(* CODESYS project Cartesin.export

Project tree, tasks and I/O mapping:
  program Cartesin [ST]
*)

// Cartesin
PROGRAM Cartesin
VAR
	Enable : BOOL;
	StartMov : BOOL;
	safe_pos :  ARRAY [1..6] OF REAL := [0.0, 0.0, 0.0, 0.0, -90.0, 0.0];
	FirstReachPos :  ARRAY [1..6] OF REAL := [0.4, 0.1, 0.606, 180, 180.000, -0.0];
	SecondReachPos :  ARRAY [1..6] OF REAL := [0.4, -0.1, 0.606, 180, 180.000, -0.0];
	FirstPerPos :  ARRAY [1..6] OF REAL := [0.4, 0.1, 0.636, 180, 180.000, -0.0];
	SecondPerPos :  ARRAY [1..6] OF REAL := [0.4, -0.1, 0.636, 180, 180.000, -0.0];
	
	CurrentPos : REAL;
	Vel : REAL := 0.5;
	Acc : REAL := 1.5;
	Jerk : REAL := 4.5;
	safepoint_overfeed : INT := 5; 
	GrRelCorner :REAL := 0.5;
	MovGroup : INT := 0;
	
	MovErr : BOOL;
	
	PowBlk : AuxAxis_PowerOn;
	PowDone, PowErr : BOOL;
	
	MovState : INT;
	InitialMov : ArcaLibrary.MCAT_MoveDirect;;
	Movs : ARRAY [0..6] OF ArcaLibrary.MC_MoveLinearAbsolute;
	StopMov : ArcaLibrary.MC_GroupStop;
	dis_trig : r_trig;
	stopEnb: BOOL;
	
	// six axis IO, Button function management
	DIp : Digital_Input;
	DOp : Digital_Output;
	enb_Timer : ton;
	enb_Delay_Time : TIME := T#1S;
	
END_VAR

// IO management
Dip(enable := TRUE);
DOP(enable := TRUE);

IF dip.DI_01 THEN	// enb button manage
	enb_Timer(in:= TRUE, pt := enb_Delay_Time); // if button has been push more then 2s
	IF enb_timer.Q AND NOT enable THEN	// enable robot
		enb_Timer(in:= FALSE);
		enable := TRUE;
	ELSIF enb_timer.Q AND enable THEN	// disable robot
		enb_Timer(in:= FALSE);
		enable := FALSE;
	END_IF
ELSE
	enb_Timer(in:= FALSE);
END_IF

IF dip.DI_02 THEN // if start button has been pressed then start mov robot
	startMov := TRUE;
END_IF

IF NOT dip.DI_03 THEN // if stop button has been pressed then stop move robot
	startMov := FALSE;
END_IF

DOp(DO_07 := PowDone);	// if robot enabled then light on

PowBlk(Enable := enable, done => PowDone);

dis_trig(clk := NOT startMov);
IF dis_trig.Q THEN
	stopEnb := TRUE;
END_IF
StopMov(AxesGroup := MovGroup, execute := stopEnb AND NOT stopmov.Done, Deceleration := vel*100, jerk := vel*1000, BufferMode := mcAborting);
IF stopmov.Done OR NOT enable THEN
	stopEnb := FALSE;	
END_IF

IF MovState > 20 AND NOT startMov THEN
	MovState := 20;
END_IF

CASE MovState OF
	0:
		IF PowDone THEN
			MovState := 10;
		END_IF
	10:
		IF startMov THEN
			MovState := 20;
		END_IF
	20:
		InitialMov(axesgroup := MovGroup, execute := FALSE);
		Movs[0](axesgroup := MovGroup, Execute := FALSE);
		Movs[1](axesgroup := MovGroup, Execute := FALSE);
		Movs[2](axesgroup := MovGroup, Execute := FALSE);
		Movs[3](axesgroup := MovGroup, Execute := FALSE);
		Movs[4](axesgroup := MovGroup, Execute := FALSE);
		Movs[5](axesgroup := MovGroup, Execute := FALSE);
		IF startMov THEN
			MovState := 30;
		ELSE
			MovState := 0;
		END_IF
	30:
		InitialMov(axesgroup := MovGroup, execute := TRUE, position := ADR(safe_pos), coordsystem := mcacs
			, BufferMode:=mcAborting, TransitionMode:= tmNone, TransitionParameter:= ADR(GrRelCorner) 
			, OverFeedPerc:= safepoint_overfeed);
		IF initialmov.Done THEN
			MovState := 40;
		END_IF
	40:
		IF Movs[4].Done THEN
			Movs[5](axesgroup := MovGroup, Execute := TRUE, Position := ADR(SecondPerPos)
				, Velocity := vel, Acceleration := acc, Deceleration := Acc, jerk := jerk
				, coordsystem := mcMcs, BufferMode := mcBlendingNext
				, TransitionMode := TMcornerdistance, TransitionParameter:=ADR(GrRelCorner)
				, Error => MovErr);
		END_IF
		Movs[0](axesgroup := MovGroup, Execute := TRUE, Position := ADR(FirstPerPos)
			, Velocity := vel, Acceleration := acc, Deceleration := Acc, jerk := jerk
			, coordsystem := mcMcs, BufferMode := mcBlendingNext
			, TransitionMode := TMcornerdistance, TransitionParameter:=ADR(GrRelCorner)
			, Error => MovErr);
		Movs[1](axesgroup := MovGroup, Execute := TRUE, Position := ADR(FirstReachPos)
			, Velocity := vel, Acceleration := acc, Deceleration := Acc, jerk := jerk
			, coordsystem := mcMcs, BufferMode := mcBlendingPrev
			, TransitionMode := TMcornerdistance, TransitionParameter:=ADR(GrRelCorner)
			, Error => MovErr);
		IF Movs[1].Done THEN
			Movs[2](axesgroup := MovGroup, Execute := FALSE);
			Movs[3](axesgroup := MovGroup, Execute := FALSE);
			Movs[4](axesgroup := MovGroup, Execute := FALSE);
			MovState := 50;
		END_IF
	50:
		Movs[2](axesgroup := MovGroup, Execute := TRUE, Position := ADR(FirstPerPos)
			, Velocity := vel, Acceleration := acc, Deceleration := Acc, jerk := jerk
			, coordsystem := mcMcs, BufferMode := mcBlendingNext
			, TransitionMode := TMcornerdistance, TransitionParameter:=ADR(GrRelCorner)
			, Error => MovErr);
		Movs[3](axesgroup := MovGroup, Execute := TRUE, Position := ADR(SecondPerPos)
			, Velocity := vel, Acceleration := acc, Deceleration := Acc, jerk := jerk
			, coordsystem := mcMcs, BufferMode := mcBlendingNext
			, TransitionMode := TMcornerdistance, TransitionParameter:=ADR(GrRelCorner)
			, Error => MovErr);
		Movs[4](axesgroup := MovGroup, Execute := TRUE, Position := ADR(SecondReachPos)
			, Velocity := vel, Acceleration := acc, Deceleration := Acc, jerk := jerk
			, coordsystem := mcMcs, BufferMode := mcBlendingPrev
			, TransitionMode := TMcornerdistance, TransitionParameter:=ADR(GrRelCorner)
			, Error => MovErr);
		IF Movs[4].Done THEN
			Movs[0](axesgroup := MovGroup, Execute := FALSE);
			Movs[1](axesgroup := MovGroup, Execute := FALSE);
			Movs[5](axesgroup := MovGroup, Execute := FALSE);
			MovState := 40;
		END_IF
END_CASE

END_PROGRAM
